// TIA Portal V19 export
FUNCTION_BLOCK "Storage"   // FB2, LAD
{ S7_Optimized_Access := 'TRUE' }
// V.0.1.0 - Created function block
// stored: MemoryReserve 100, SetENOAutomatically false
   VAR_INPUT
      Insert_Item : Int;   // Insert item type into storage
      Take_Item : Int;   // Remove item type from storage
      Storage_Max : Int := 5;   // Maximum storage amount allowed
      Storage_Min : Int := 3;   // Minimum storage amount after production
   END_VAR
   VAR_OUTPUT
      Storage_1 : Int;   // How many items are currently on space A
      Storage_2 : Int;   // How many items are currently on space B
      Storage_3 : Int;   // How many items are currently on space C
   END_VAR
   VAR
      Items_On_Space_1 : Int;   // Amount of items on space 1
      Items_On_Space_2 : Int;   // Amount of items on space 2
      Items_On_Space_3 : Int;   // Amount of items on space 3
   END_VAR
BEGIN

REGION Network 1: Insert items into storage
   // If inserting type X, then check if capacity is reached. If below full capacity then add item
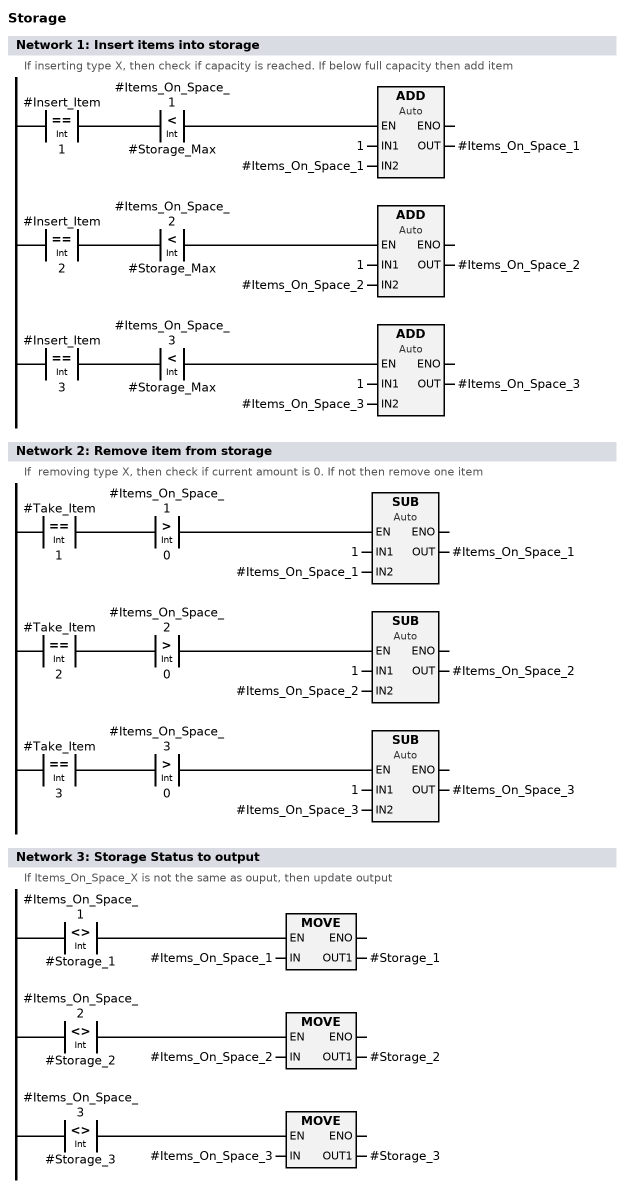
   RUNG wire#powerrail
      { S7_Templates := "SrcType := Int" } EQ_Contact(in1 := #Insert_Item, in2 := 1)
      { S7_Templates := "SrcType := Int" } LT_Contact(in1 := #Items_On_Space_1, in2 := #Storage_Max)
      Add(in1 := 1, in2 := #Items_On_Space_1, out => #Items_On_Space_1)
   END_RUNG
   RUNG wire#powerrail
      { S7_Templates := "SrcType := Int" } EQ_Contact(in1 := #Insert_Item, in2 := 2)
      { S7_Templates := "SrcType := Int" } LT_Contact(in1 := #Items_On_Space_2, in2 := #Storage_Max)
      Add(in1 := 1, in2 := #Items_On_Space_2, out => #Items_On_Space_2)
   END_RUNG
   RUNG wire#powerrail
      { S7_Templates := "SrcType := Int" } EQ_Contact(in1 := #Insert_Item, in2 := 3)
      { S7_Templates := "SrcType := Int" } LT_Contact(in1 := #Items_On_Space_3, in2 := #Storage_Max)
      Add(in1 := 1, in2 := #Items_On_Space_3, out => #Items_On_Space_3)
   END_RUNG
   // the same network as SCL:
   IF (#Insert_Item = 1) AND (#Items_On_Space_1 < #Storage_Max) THEN
       #Items_On_Space_1 := 1 + #Items_On_Space_1;
   END_IF;
   IF (#Insert_Item = 2) AND (#Items_On_Space_2 < #Storage_Max) THEN
       #Items_On_Space_2 := 1 + #Items_On_Space_2;
   END_IF;
   IF (#Insert_Item = 3) AND (#Items_On_Space_3 < #Storage_Max) THEN
       #Items_On_Space_3 := 1 + #Items_On_Space_3;
   END_IF;
END_REGION

REGION Network 2: Remove item from storage
   // If  removing type X, then check if current amount is 0. If not then remove one item
   RUNG wire#powerrail
      { S7_Templates := "SrcType := Int" } EQ_Contact(in1 := #Take_Item, in2 := 1)
      { S7_Templates := "SrcType := Int" } GT_Contact(in1 := #Items_On_Space_1, in2 := 0)
      Sub(in1 := 1, in2 := #Items_On_Space_1, out => #Items_On_Space_1)
   END_RUNG
   RUNG wire#powerrail
      { S7_Templates := "SrcType := Int" } EQ_Contact(in1 := #Take_Item, in2 := 2)
      { S7_Templates := "SrcType := Int" } GT_Contact(in1 := #Items_On_Space_2, in2 := 0)
      Sub(in1 := 1, in2 := #Items_On_Space_2, out => #Items_On_Space_2)
   END_RUNG
   RUNG wire#powerrail
      { S7_Templates := "SrcType := Int" } EQ_Contact(in1 := #Take_Item, in2 := 3)
      { S7_Templates := "SrcType := Int" } GT_Contact(in1 := #Items_On_Space_3, in2 := 0)
      Sub(in1 := 1, in2 := #Items_On_Space_3, out => #Items_On_Space_3)
   END_RUNG
   // the same network as SCL:
   IF (#Take_Item = 1) AND (#Items_On_Space_1 > 0) THEN #Items_On_Space_1 := 1 - #Items_On_Space_1; END_IF;
   IF (#Take_Item = 2) AND (#Items_On_Space_2 > 0) THEN #Items_On_Space_2 := 1 - #Items_On_Space_2; END_IF;
   IF (#Take_Item = 3) AND (#Items_On_Space_3 > 0) THEN #Items_On_Space_3 := 1 - #Items_On_Space_3; END_IF;
END_REGION

REGION Network 3: Storage Status to output
   // If Items_On_Space_X is not the same as ouput, then update output
   RUNG wire#powerrail
      { S7_Templates := "SrcType := Int" } NE_Contact(in1 := #Items_On_Space_1, in2 := #Storage_1)
      Move(in := #Items_On_Space_1, out1 => #Storage_1)
   END_RUNG
   RUNG wire#powerrail
      { S7_Templates := "SrcType := Int" } NE_Contact(in1 := #Items_On_Space_2, in2 := #Storage_2)
      Move(in := #Items_On_Space_2, out1 => #Storage_2)
   END_RUNG
   RUNG wire#powerrail
      { S7_Templates := "SrcType := Int" } NE_Contact(in1 := #Items_On_Space_3, in2 := #Storage_3)
      Move(in := #Items_On_Space_3, out1 => #Storage_3)
   END_RUNG
   // the same network as SCL:
   IF #Items_On_Space_1 <> #Storage_1 THEN #Storage_1 := #Items_On_Space_1; END_IF;
   IF #Items_On_Space_2 <> #Storage_2 THEN #Storage_2 := #Items_On_Space_2; END_IF;
   IF #Items_On_Space_3 <> #Storage_3 THEN #Storage_3 := #Items_On_Space_3; END_IF;
END_REGION
END_FUNCTION_BLOCK
